{region '#Template'}
	{attribute 'Version' := '5.0.0.0'}
	{attribute 'Tags' := '"LCID": "1031", "Text": "Automatisierungssteuerung, Gerät, Einstellungen, Projekt, Parameter"'}
	{attribute 'Tags' := '"LCID": "1033", "Text": "Automation control, Device, Settings, Project, Parameter"'}
	{attribute 'Description' := '"LCID": "1031", "Text": "Basis Parameter"'}
	{attribute 'Description' := '"LCID": "1033", "Text": "Basic settings"'}
{endregion}

FUNCTION_BLOCK FB_BA_Parameter
VAR_INPUT
END_VAR
VAR_OUTPUT
END_VAR
VAR		
//		Recipient		: FB_BACnet_RcpList;	
END_VAR

// Recipient list to write (to all event classes):
// Recipient();

METHOD FB_init : BOOL
VAR_INPUT
	bInitRetains : BOOL; // if TRUE, the retain variables are initialized (warm start / cold start)
	bInCopyCode : BOOL;  // if TRUE, the instance afterwards gets moved into the copy code (online change)
END_VAR
VAR
	Parameters 				: FB_BA_Param;	
END_VAR
//Writeaccess on EventEnable Bits (Property 35.)
Parameters.SetDefWriteAccess(E_BA_Parameter.eEventEnable, E_BA_ROLE.eInternal);

//DefaultSeparator on each DPAD Level
Parameters.DPAD_ObjectName_DefSeparator:='-';
Parameters.DPAD_Description_DefSeparator:=' - ';

//Default structure of BACnetObjects in Systemmanager 
Parameters.BACnet_View_SubordinateAnnotationMode := Tc3_BACnetRev14.E_BACnet_AnnotationTitle.eObjectName;

//Set AckknowledgeRequiredFlags to AMEV 2017 Standard (Property 1.)
Parameters.AckFlags_Simple 		:= F_BA_EventTransition(bToOffNormal:= FALSE, bToFault:=FALSE, bToNormal:=FALSE);
Parameters.AckFlags_Standard	:= F_BA_EventTransition(bToOffNormal:= TRUE, bToFault:=FALSE, bToNormal:=FALSE);
Parameters.AckFlags_Extended 	:= F_BA_EventTransition(bToOffNormal:= TRUE, bToFault:=FALSE, bToNormal:=TRUE);

//Set EventEnable to AMEV 2017 Standard (Property 35.)
Parameters.EventEn_Simple 		:= F_BA_EventTransition(bToOffNormal:= TRUE, bToFault:=FALSE, bToNormal:=TRUE);
Parameters.EventEn_Standard		:= F_BA_EventTransition(bToOffNormal:= TRUE, bToFault:=FALSE, bToNormal:=TRUE);
Parameters.EventEn_Extended		:= F_BA_EventTransition(bToOffNormal:= TRUE, bToFault:=FALSE, bToNormal:=TRUE);

// Quittier- und Rücksetzmodus	// Acknowledge mode
// E_BA_AcknowledgeMode.eSingle	// Acknowledges only the next outstanding event transition by executing an acknowledgement.
// E_BA_AcknowledgeMode.eEntire	// Acknowledges all unacknowledged event transitions by executing a single acknowledgement.
Parameters.EvtMgmt_AckMode		:= E_BA_AcknowledgeMode.eSingle;
END_METHOD

END_FUNCTION_BLOCK

(* stored: Version 1.1.0.1, ProductVersion 3.1.4024.12
   POU FB_BA_Parameter: Id {78edb545-3849-4eb5-9deb-c438d7453294}, SpecialFunc None
   Method FB_init: Id {6ffd1bdd-8fda-48ba-891d-8d275c66517c} *)
